{attribute addProperty BoxType "EL6201-0000-0017"}
{attribute addProperty Id "ASI_Inputs_DeviceAT %I*ASI_Inputs_Device_6E2FC913248310ASI_StatusAT %I*ASI_Status_A408178488110ASI_Outputs_DeviceAT %Q*ASI_Outputs_Device_4A17E548248310ASI_ControlAT %Q*ASI_Control_3C9D221D4050WcStateAT %I*WcState_F855686C1620InfoDataAT %I*InfoData_BC63D37F80100"}
{attribute addProperty CRC "1178315670"}
{attribute addProperty SizeInBites "720"}
{attribute addProperty SizeInBytes "90"}
TYPE EL6201_34DED8B9 :
STRUCT
	{attribute addProperty Name "ASI_Inputs_Device"}
	ASI_Inputs_Device : ASI_Inputs_Device_6E2FC913;
	{attribute addProperty Name "ASI_Status"}
	ASI_Status : ASI_Status_A4081784;
	{attribute addProperty Name "ASI_Outputs_Device"}
	ASI_Outputs_Device : ASI_Outputs_Device_4A17E548;
	{attribute addProperty Name "ASI_Control"}
	ASI_Control : ASI_Control_3C9D221D;
	{attribute addProperty Name "WcState"}
	WcState : WcState_F855686C;
	{attribute addProperty Name "InfoData"}
	InfoData : InfoData_BC63D37F;
END_STRUCT
END_TYPE

(* stored: Version 1.2.0.0, ProductVersion 3.1.4024.9
   DUT EL6201_34DED8B9: Id {1c64582a-1e05-4625-8b77-7ad128f8d891} *)
